(* IEC 61131-3 sources: router_agent/backend/app/tests/eval/formal_st_files, 10 files *)

(* ---- example_y_equals_x.st ---- *)
FUNCTION_BLOCK Example
VAR_INPUT
    x : BOOL;
END_VAR
VAR_OUTPUT
    y : BOOL;
END_VAR

y := x;

//#ASSERT (y = x) : assert_y_equals_x
END_FUNCTION_BLOCK

(* ---- fb_and2_output.st ---- *)
FUNCTION_BLOCK FB_And2
VAR_INPUT
    a : BOOL;
    b : BOOL;
END_VAR
VAR_OUTPUT
    y : BOOL;
END_VAR

y := a AND b;

//#ASSERT (y = (a AND b)) : assert_y_is_a_and_b
END_FUNCTION_BLOCK

(* ---- fb_fault_dominates.st ---- *)
FUNCTION_BLOCK FB_FaultDominates
VAR_INPUT
    enable : BOOL;
    fault : BOOL;
END_VAR
VAR_OUTPUT
    run : BOOL;
END_VAR

run := enable AND NOT fault;

//#ASSERT (run = (enable AND NOT fault)) : assert_run_respects_fault
END_FUNCTION_BLOCK

(* ---- fb_imp_alarm_follows_sensor.st ---- *)
FUNCTION_BLOCK FB_Imp
VAR_INPUT
    sensor : BOOL;
END_VAR
VAR_OUTPUT
    alarm : BOOL;
END_VAR

alarm := sensor;

//#ASSERT (alarm = sensor) : assert_alarm_follows_sensor
END_FUNCTION_BLOCK

(* ---- fb_limit_protect.st ---- *)
FUNCTION_BLOCK FB_LimitProtect
VAR_INPUT
    command : BOOL;
    limit : BOOL;
END_VAR
VAR_OUTPUT
    move : BOOL;
END_VAR

move := command AND NOT limit;

//#ASSERT (move = (command AND NOT limit)) : assert_move_respects_limit
END_FUNCTION_BLOCK

(* ---- fb_mode_mux.st ---- *)
FUNCTION_BLOCK FB_ModeMux
VAR_INPUT
    autoMode : BOOL;
    manualCmd : BOOL;
    autoCmd : BOOL;
END_VAR
VAR_OUTPUT
    outputCmd : BOOL;
END_VAR

outputCmd := (autoMode AND autoCmd) OR ((NOT autoMode) AND manualCmd);

//#ASSERT (outputCmd = ((autoMode AND autoCmd) OR ((NOT autoMode) AND manualCmd))) : assert_mode_selects_command
END_FUNCTION_BLOCK

(* ---- fb_mutex_outputs.st ---- *)
FUNCTION_BLOCK FB_MutexOutputs
VAR_INPUT
    fwd : BOOL;
    rev : BOOL;
END_VAR
VAR_OUTPUT
    forward : BOOL;
    reverse : BOOL;
END_VAR

forward := fwd AND NOT rev;
reverse := rev AND NOT fwd;

//#ASSERT (NOT (forward AND reverse)) : assert_forward_reverse_mutex
END_FUNCTION_BLOCK

(* ---- fb_not_output.st ---- *)
FUNCTION_BLOCK FB_NotOutput
VAR_INPUT
    x : BOOL;
END_VAR
VAR_OUTPUT
    y : BOOL;
END_VAR

y := NOT x;

//#ASSERT (y = NOT x) : assert_y_is_not_x
END_FUNCTION_BLOCK

(* ---- fb_or2_output.st ---- *)
FUNCTION_BLOCK FB_Or2
VAR_INPUT
    a : BOOL;
    b : BOOL;
END_VAR
VAR_OUTPUT
    y : BOOL;
END_VAR

y := a OR b;

//#ASSERT (y = (a OR b)) : assert_y_is_a_or_b
END_FUNCTION_BLOCK

(* ---- fb_stop_dominates.st ---- *)
FUNCTION_BLOCK FB_StopDominates
VAR_INPUT
    start : BOOL;
    stop : BOOL;
END_VAR
VAR_OUTPUT
    motor : BOOL;
END_VAR

motor := start AND NOT stop;

//#ASSERT (motor = (start AND NOT stop)) : assert_motor_respects_stop
END_FUNCTION_BLOCK
